  TelegramState.UNDEFINED                : TELEGRAM_STATE_TO_STRING := StrReplace('UNDEFINED ({0})'               ,'{0}', USINT_TO_STRING(State));
  TelegramState.ERROR_161                : TELEGRAM_STATE_TO_STRING := StrReplace('ERROR_161 ({0})'               ,'{0}', USINT_TO_STRING(State));
  TelegramState.ERROR_162                : TELEGRAM_STATE_TO_STRING := StrReplace('ERROR_162 ({0})'               ,'{0}', USINT_TO_STRING(State));
  TelegramState.ERROR_163                : TELEGRAM_STATE_TO_STRING := StrReplace('ERROR_163 ({0})'               ,'{0}', USINT_TO_STRING(State));
  TelegramState.ERROR_164                : TELEGRAM_STATE_TO_STRING := StrReplace('ERROR_164 ({0})'               ,'{0}', USINT_TO_STRING(State));
  TelegramState.ERROR_165                : TELEGRAM_STATE_TO_STRING := StrReplace('ERROR_165 ({0})'               ,'{0}', USINT_TO_STRING(State));
  TelegramState.ERROR_166                : TELEGRAM_STATE_TO_STRING := StrReplace('ERROR_166 ({0})'               ,'{0}', USINT_TO_STRING(State));
  TelegramState.ERROR_167                : TELEGRAM_STATE_TO_STRING := StrReplace('ERROR_167 ({0})'               ,'{0}', USINT_TO_STRING(State));
  TelegramState.ERROR_168                : TELEGRAM_STATE_TO_STRING := StrReplace('ERROR_168 ({0})'               ,'{0}', USINT_TO_STRING(State));
  TelegramState.ERROR_169                : TELEGRAM_STATE_TO_STRING := StrReplace('ERROR_169 ({0})'               ,'{0}', USINT_TO_STRING(State));
  TelegramState.ERROR_170                : TELEGRAM_STATE_TO_STRING := StrReplace('ERROR_170 ({0})'               ,'{0}', USINT_TO_STRING(State));
  TelegramState.ERROR_171                : TELEGRAM_STATE_TO_STRING := StrReplace('ERROR_171 ({0})'               ,'{0}', USINT_TO_STRING(State));
  TelegramState.ERROR_172                : TELEGRAM_STATE_TO_STRING := StrReplace('ERROR_172 ({0})'               ,'{0}', USINT_TO_STRING(State));
  TelegramState.READY_TO_RESUME          : TELEGRAM_STATE_TO_STRING := StrReplace('READY_TO_RESUME ({0})'         ,'{0}', USINT_TO_STRING(State));
  TelegramState.READY_FOR_INITIALIZATION : TELEGRAM_STATE_TO_STRING := StrReplace('READY_FOR_INITIALIZATION ({0})','{0}', USINT_TO_STRING(State));
  TelegramState.INITIALIZED              : TELEGRAM_STATE_TO_STRING := StrReplace('INITIALIZED ({0})'             ,'{0}', USINT_TO_STRING(State));  
ELSE
  TELEGRAM_STATE_TO_STRING := CONCAT('TelegramStateToString-Function: Error -> no parsing for value ', USINT_TO_STRING(State));
END_CASE

END_FUNCTION

// Library/Functions/Convert/TO_STRING/THRESHOLD_MODE_TO_STRING
FUNCTION THRESHOLD_MODE_TO_STRING : STRING
// ------------------------------------------------------------------------- 
//  SRCI Robot Library                                                
// ------------------------------------------------------------------------- 
//                                                                           
//  Object:      THRESHOLD_MODE_TO_STRING                                       
//  Author:      Thorsten Brach                                                
//  Date:        2025-01-24
//
//  Description:                                              
//   
//                                                                           
//  Copyright: 
//    (C) 2025 Thorsten Brach. All rights reserved                                                                                                                                            
//             Licensed under the LGPL-3.0 license.
//                                                                           
//  Disclaimer:                                                                           
//    This project is provided without any guarantee and can be used for   
//    private and commercial purposes. Any use is at the user’s 
//    own risk and responsibility.
//
// -------------------------------------------------------------------------
VAR_INPUT
  /// ThresholdMode
  Value : ThresholdMode;
END_VAR

CASE Value 
OF

  ThresholdMode.AUTOMATIC : StrReplace('AUTOMATIC ({0})','{0}' , USINT_TO_STRING(Value));
  ThresholdMode.MANUAL    : StrReplace('MANUAL ({0})'   ,'{0}' , USINT_TO_STRING(Value));

END_CASE

END_FUNCTION

// Library/Functions/Convert/TO_STRING/TOOL_CALCULATION_MODE_TO_STRING
FUNCTION TOOL_CALCULATION_MODE_TO_STRING : STRING
// ------------------------------------------------------------------------- 
//  SRCI Robot Library                                                
// ------------------------------------------------------------------------- 
//                                                                           
//  Object:      TOOL_CALCULATION_MODE_TO_STRING                                       
//  Author:      Thorsten Brach                                                
//  Date:        2025-02-01
//
//  Description:                                              
//   
//                                                                           
//  Copyright: 
//    (C) 2025 Thorsten Brach. All rights reserved                                                                                                                                            
//             Licensed under the LGPL-3.0 license.
//                                                                           
//  Disclaimer:                                                                           
//    This project is provided without any guarantee and can be used for   
//    private and commercial purposes. Any use is at the user’s 
//    own risk and responsibility.
//
// -------------------------------------------------------------------------
VAR_INPUT
  /// ToolCalculationMode
  Value : ToolCalculationMode;
END_VAR

CASE Value 
OF

  ToolCalculationMode.TWO_POINT_Z_METHOD   : StrReplace('TWO_POINT_Z_METHOD ({0})'  ,'{0}' , SINT_TO_STRING(Value));
  ToolCalculationMode.THREE_POINT_METHOD   : StrReplace('THREE_POINT_METHOD ({0})'  ,'{0}' , SINT_TO_STRING(Value));
  ToolCalculationMode.FOUR_POINT_METHOD    : StrReplace('FOUR_POINT_METHOD ({0})'   ,'{0}' , SINT_TO_STRING(Value));
  ToolCalculationMode.FIVE_POINT_METHOD    : StrReplace('FIVE_POINT_METHOD ({0})'   ,'{0}' , SINT_TO_STRING(Value));
  ToolCalculationMode.SIX_POINT_METHOD     : StrReplace('SIX_POINT_METHOD ({0})'    ,'{0}' , SINT_TO_STRING(Value));
  ToolCalculationMode.ABC_WORLD_METHOD     : StrReplace('ABC_WORLD_METHOD ({0})'    ,'{0}' , SINT_TO_STRING(Value));
  ToolCalculationMode.ABC_TWO_POINT_METHOD : StrReplace('ABC_TWO_POINT_METHOD ({0})','{0}' , SINT_TO_STRING(Value));
  
END_CASE

END_FUNCTION

// Library/Functions/Convert/TO_STRING/TRANSFORM_MODE_TO_STRING
FUNCTION TRANSFORM_MODE_TO_STRING : STRING
// ------------------------------------------------------------------------- 
//  SRCI Robot Library                                                
// ------------------------------------------------------------------------- 
//                                                                           
//  Object:      TRANSFORM_MODE_TO_STRING                                       
//  Author:      Thorsten Brach                                                
//  Date:        2025-01-24
//
//  Description:                                              
//   
//                                                                           
//  Copyright: 
//    (C) 2025 Thorsten Brach. All rights reserved                                                                                                                                            
//             Licensed under the LGPL-3.0 license.
//                                                                           
//  Disclaimer:                                                                           
//    This project is provided without any guarantee and can be used for   
//    private and commercial purposes. Any use is at the user’s 
//    own risk and responsibility.
//
// -------------------------------------------------------------------------
VAR_INPUT
  /// TransformMode
  Value : TransformMode;
END_VAR

CASE Value 
OF

  TransformMode.MIRROR_AT_POINT             : StrReplace('MIRROR_AT_POINT ({0})'             ,'{0}' , SINT_TO_STRING(Value));
  TransformMode.MIRROR_AT_STRAIGHT_LINE     : StrReplace('MIRROR_AT_STRAIGHT_LINE ({0})'     ,'{0}' , SINT_TO_STRING(Value));
  TransformMode.MIRROR_AT_PLANE             : StrReplace('MIRROR_AT_PLANE ({0})'             ,'{0}' , SINT_TO_STRING(Value));
  TransformMode.ROTATE_AROUND_STRAIGHT_LINE : StrReplace('ROTATE_AROUND_STRAIGHT_LINE ({0})' ,'{0}' , SINT_TO_STRING(Value));
  TransformMode.SHIFT_BY_VECTOR             : StrReplace('SHIFT_BY_VECTOR ({0})'             ,'{0}' , SINT_TO_STRING(Value));

END_CASE

END_FUNCTION

// Library/Functions/Convert/TO_STRING/TRIGGER_CONDITION_TO_STRING
FUNCTION TRIGGER_CONDITION_TO_STRING : STRING
// ------------------------------------------------------------------------- 
//  SRCI Robot Library                                                
// ------------------------------------------------------------------------- 
//                                                                           
//  Object:      TRIGGER_CONDITION_TO_STRING                                       
//  Author:      Thorsten Brach                                                
//  Date:        2025-02-01
//
//  Description:                                              
//   
//                                                                           
//  Copyright: 
//    (C) 2025 Thorsten Brach. All rights reserved                                                                                                                                            
//             Licensed under the LGPL-3.0 license.
//                                                                           
//  Disclaimer:                                                                           
//    This project is provided without any guarantee and can be used for   
//    private and commercial purposes. Any use is at the user’s 
//    own risk and responsibility.
//
// -------------------------------------------------------------------------
VAR_INPUT
  /// TriggerCondition
  Value : TriggerCondition;
END_VAR

CASE Value 
OF

  TriggerCondition.TARGET_POSITION_TIME_MS                : StrReplace('TARGET_POSITION_TIME_MS ({0})'               ,'{0}' , SINT_TO_STRING(Value));
  TriggerCondition.TARGET_POSITION_TCP_VELOCITY_ABSOLUTE  : StrReplace('TARGET_POSITION_TCP_VELOCITY_ABSOLUTE ({0})' ,'{0}' , SINT_TO_STRING(Value));
  TriggerCondition.TARGET_POSITION_TCP_VELOCITY_PERCENT   : StrReplace('TARGET_POSITION_TCP_VELOCITY_PERCENT ({0})'  ,'{0}' , SINT_TO_STRING(Value));
  TriggerCondition.TARGET_POSITION_DISTANCE_ABSOLUTE      : StrReplace('TARGET_POSITION_DISTANCE_ABSOLUTE ({0})'     ,'{0}' , SINT_TO_STRING(Value));
  TriggerCondition.TARGET_POSITION_DISTANCE_PERCENT       : StrReplace('TARGET_POSITION_DISTANCE_PERCENT ({0})'      ,'{0}' , SINT_TO_STRING(Value));
  TriggerCondition.UNDEFINED                              : StrReplace('UNDEFINED ({0})'                             ,'{0}' , SINT_TO_STRING(Value));
  TriggerCondition.START_POSITION_DISTANCE_PERCENT        : StrReplace('START_POSITION_DISTANCE_PERCENT ({0})'       ,'{0}' , SINT_TO_STRING(Value));
  TriggerCondition.START_POSITION_DISTANCE_ABSOLUTE       : StrReplace('START_POSITION_DISTANCE_ABSOLUTE ({0})'      ,'{0}' , SINT_TO_STRING(Value));
  TriggerCondition.START_POSITION_TCP_VELOCITY_PERCENT    : StrReplace('START_POSITION_TCP_VELOCITY_PERCENT ({0})'   ,'{0}' , SINT_TO_STRING(Value));
  TriggerCondition.START_POSITION_TCP_VELOCIT_ABSOLUTE    : StrReplace('START_POSITION_TCP_VELOCIT_ABSOLUTE ({0})'   ,'{0}' , SINT_TO_STRING(Value));
  TriggerCondition.START_POSITION_TIME_MS                 : StrReplace('START_POSITION_TCP_VELOCIT_ABSOLUTE ({0})'   ,'{0}' , SINT_TO_STRING(Value));

END_CASE

END_FUNCTION

// Library/Functions/Convert/TO_STRING/TRIGGER_MODE_IO_TO_STRING
FUNCTION TRIGGER_MODE_IO_TO_STRING : STRING
// ------------------------------------------------------------------------- 
//  SRCI Robot Library                                                
// ------------------------------------------------------------------------- 
//                                                                           
//  Object:      TRIGGER_MODE_IO_TO_STRING                                       
//  Author:      Thorsten Brach                                                
//  Date:        2025-02-01
//
//  Description:                                              
//   
//                                                                           
//  Copyright: 
//    (C) 2025 Thorsten Brach. All rights reserved                                                                                                                                            
//             Licensed under the LGPL-3.0 license.
//                                                                           
//  Disclaimer:                                                                           
//    This project is provided without any guarantee and can be used for   
//    private and commercial purposes. Any use is at the user’s 
//    own risk and responsibility.
//
// -------------------------------------------------------------------------
VAR_INPUT
  /// TriggerModeIo
  Value : TriggerModeIo;
END_VAR

CASE Value 
OF

  TriggerModeIo.INVALID                                                             : StrReplace('INVALID ({0})'                                                              ,'{0}' , SINT_TO_STRING(Value));
  TriggerModeIo.DIGITAL_INPUT_RISING_EDGE                                           : StrReplace('DIGITAL_INPUT_RISING_EDGE ({0})'                                            ,'{0}' , SINT_TO_STRING(Value));
  TriggerModeIo.DIGITAL_INPUT_FALLING_EDGE                                          : StrReplace('DIGITAL_INPUT_FALLING_EDGE ({0})'                                           ,'{0}' , SINT_TO_STRING(Value));
  TriggerModeIo.DIGITAL_INPUT_RISING_OR_FALLING_EDGE                                : StrReplace('DIGITAL_INPUT_RISING_OR_FALLING_EDGE ({0})'                                 ,'{0}' , SINT_TO_STRING(Value));
  TriggerModeIo.DIGITAL_INPUT_RISING_OR_FALLING_EDGE_INVERTED                       : StrReplace('DIGITAL_INPUT_RISING_OR_FALLING_EDGE_INVERTED ({0})'                        ,'{0}' , SINT_TO_STRING(Value));
  TriggerModeIo.DIGITAL_OUTPUT_RISING_EDGE                                          : StrReplace('DIGITAL_OUTPUT_RISING_EDGE ({0})'                                           ,'{0}' , SINT_TO_STRING(Value));
  TriggerModeIo.DIGITAL_OUTPUT_FALLING_EDGE                                         : StrReplace('DIGITAL_OUTPUT_FALLING_EDGE ({0})'                                          ,'{0}' , SINT_TO_STRING(Value));
  TriggerModeIo.DIGITAL_OUTPUT_RISING_OR_FALLING_EDGE                               : StrReplace('DIGITAL_OUTPUT_RISING_OR_FALLING_EDGE ({0})'                                ,'{0}' , SINT_TO_STRING(Value));
  TriggerModeIo.DIGITAL_OUTPUT_RISING_OR_FALLING_EDGE_INVERTED                      : StrReplace('DIGITAL_OUTPUT_RISING_OR_FALLING_EDGE_INVERTED ({0})'                       ,'{0}' , SINT_TO_STRING(Value));
  TriggerModeIo.ANALOG_INPUT_EXCEEDING_DEFINED_THRESHOLD                            : StrReplace('ANALOG_INPUT_EXCEEDING_DEFINED_THRESHOLD ({0})'                             ,'{0}' , SINT_TO_STRING(Value));
  TriggerModeIo.ANALOG_INPUT_FALLING_BELOW_DEFINED_THRESHOLD                        : StrReplace('ANALOG_INPUT_FALLING_BELOW_DEFINED_THRESHOLD ({0})'                         ,'{0}' , SINT_TO_STRING(Value));
  TriggerModeIo.ANALOG_INPUT_EXCEEDING_OR_FALLING_BELOW_DEFINED_THRESHOLD           : StrReplace('ANALOG_INPUT_EXCEEDING_OR_FALLING_BELOW_DEFINED_THRESHOLD ({0})'            ,'{0}' , SINT_TO_STRING(Value));
  TriggerModeIo.ANALOG_INPUT_EXCEEDING_OR_FALLING_BELOW_DEFINED_THRESHOLD_INVERTED  : StrReplace('ANALOG_INPUT_EXCEEDING_OR_FALLING_BELOW_DEFINED_THRESHOLD_INVERTED ({0})'   ,'{0}' , SINT_TO_STRING(Value));
  TriggerModeIo.ANALOG_INPUT_ENTERING_DEFINED_RANGE                                 : StrReplace('ANALOG_INPUT_ENTERING_DEFINED_RANGE ({0})'                                  ,'{0}' , SINT_TO_STRING(Value));
  TriggerModeIo.ANALOG_INPUT_LEAVING_DEFINED_RANGE                                  : StrReplace('ANALOG_INPUT_LEAVING_DEFINED_RANGE ({0})'                                   ,'{0}' , SINT_TO_STRING(Value));
  TriggerModeIo.ANALOG_INPUT_ENTERING_OR_LEAVING_DEFINED_RANGE                      : StrReplace('ANALOG_INPUT_ENTERING_OR_LEAVING_DEFINED_RANGE ({0})'                       ,'{0}' , SINT_TO_STRING(Value));
  TriggerModeIo.ANALOG_INPUT_ENTERING_OR_LEAVING_DEFINED_RANGE_INVERTED             : StrReplace('ANALOG_INPUT_ENTERING_OR_LEAVING_DEFINED_RANGE_INVERTED ({0})'              ,'{0}' , SINT_TO_STRING(Value));
  TriggerModeIo.ANALOG_OUTPUT_EXCEEDING_DEFINED_THRESHOLD                           : StrReplace('ANALOG_OUTPUT_EXCEEDING_DEFINED_THRESHOLD ({0})'                            ,'{0}' , SINT_TO_STRING(Value));
  TriggerModeIo.ANALOG_OUTPUT_FALLING_BELOW_DEFINED_THRESHOLD                       : StrReplace('ANALOG_OUTPUT_FALLING_BELOW_DEFINED_THRESHOLD ({0})'                        ,'{0}' , SINT_TO_STRING(Value));
  TriggerModeIo.ANALOG_OUTPUT_EXCEEDING_OR_FALLING_BELOW_DEFINED_THRESHOLD          : StrReplace('ANALOG_OUTPUT_EXCEEDING_OR_FALLING_BELOW_DEFINED_THRESHOLD ({0})'           ,'{0}' , SINT_TO_STRING(Value));
  TriggerModeIo.ANALOG_OUTPUT_EXCEEDING_OR_FALLING_BELOW_DEFINED_THRESHOLD_INVERTED : StrReplace('ANALOG_OUTPUT_EXCEEDING_OR_FALLING_BELOW_DEFINED_THRESHOLD_INVERTED ({0})'  ,'{0}' , SINT_TO_STRING(Value));
  TriggerModeIo.ANALOG_OUTPUT_ENTERING_DEFINED_RANGE                                : StrReplace('ANALOG_OUTPUT_ENTERING_DEFINED_RANGE ({0})'                                 ,'{0}' , SINT_TO_STRING(Value));
  TriggerModeIo.ANALOG_OUTPUT_LEAVING_DEFINED_RANGE                                 : StrReplace('ANALOG_OUTPUT_LEAVING_DEFINED_RANGE ({0})'                                  ,'{0}' , SINT_TO_STRING(Value));
  TriggerModeIo.ANALOG_OUTPUT_ENTERING_OR_LEAVING_DEFINED_RANGE                     : StrReplace('ANALOG_OUTPUT_ENTERING_OR_LEAVING_DEFINED_RANGE ({0})'                      ,'{0}' , SINT_TO_STRING(Value));
  TriggerModeIo.ANALOG_OUTPUT_ENTERING_OR_LEAVING_DEFINED_RANGE_INVERTED            : StrReplace('ANALOG_OUTPUT_ENTERING_OR_LEAVING_DEFINED_RANGE_INVERTED ({0})'             ,'{0}' , SINT_TO_STRING(Value));
  TriggerModeIo.INTEGER_REGISTER_EXCEEDING_DEFINED_THRESHOLD                        : StrReplace('INTEGER_REGISTER_EXCEEDING_DEFINED_THRESHOLD ({0})'                         ,'{0}' , SINT_TO_STRING(Value));
  TriggerModeIo.INTEGER_REGISTER_FALLING_BELOW_DEFINED_THRESHOLD                    : StrReplace('INTEGER_REGISTER_FALLING_BELOW_DEFINED_THRESHOLD ({0})'                     ,'{0}' , SINT_TO_STRING(Value));
  TriggerModeIo.INTEGER_REGISTER_EXCEEDING_OR_FALLING_BELOW_DEFINED_THRESHOLD       : StrReplace('INTEGER_REGISTER_EXCEEDING_OR_FALLING_BELOW_DEFINED_THRESHOLD ({0})'        ,'{0}' , SINT_TO_STRING(Value));
  TriggerModeIo.INTEGER_REGISTER_EXCEEDING_OR_FALLING_BELOW_DEFINED_VALUE_INVERTED  : StrReplace('INTEGER_REGISTER_EXCEEDING_OR_FALLING_BELOW_DEFINED_VALUE_INVERTED ({0})'   ,'{0}' , SINT_TO_STRING(Value));
  TriggerModeIo.INTEGER_REGISTER_ENTERING_DEFINED_RANGE                             : StrReplace('INTEGER_REGISTER_ENTERING_DEFINED_RANGE ({0})'                              ,'{0}' , SINT_TO_STRING(Value));
  TriggerModeIo.INTEGER_REGISTER_LEAVING_DEFINED_RANGE                              : StrReplace('INTEGER_REGISTER_LEAVING_DEFINED_RANGE ({0})'                               ,'{0}' , SINT_TO_STRING(Value));
  TriggerModeIo.INTEGER_REGISTER_ENTERING_OR_LEAVING_DEFINED_RANGE                  : StrReplace('INTEGER_REGISTER_ENTERING_OR_LEAVING_DEFINED_RANGE ({0})'                   ,'{0}' , SINT_TO_STRING(Value));
  TriggerModeIo.INTEGER_REGISTER_ENTERING_OR_LEAVING_DEFINED_RANGE_INVERTED         : StrReplace('INTEGER_REGISTER_ENTERING_OR_LEAVING_DEFINED_RANGE_INVERTED ({0})'          ,'{0}' , SINT_TO_STRING(Value));
  TriggerModeIo.REAL_REGISTER_EXCEEDING_DEFINED_THRESHOLD                           : StrReplace('REAL_REGISTER_EXCEEDING_DEFINED_THRESHOLD ({0})'                            ,'{0}' , SINT_TO_STRING(Value));
  TriggerModeIo.REAL_REGISTER_FALLING_BELOW_DEFINED_THRESHOLD                       : StrReplace('REAL_REGISTER_FALLING_BELOW_DEFINED_THRESHOLD ({0})'                        ,'{0}' , SINT_TO_STRING(Value));
  TriggerModeIo.REAL_REGISTER_EXCEEDING_OR_FALLING_BELOW_DEFINED_THRESHOLD          : StrReplace('REAL_REGISTER_EXCEEDING_OR_FALLING_BELOW_DEFINED_THRESHOLD ({0})'           ,'{0}' , SINT_TO_STRING(Value));
  TriggerModeIo.REAL_REGISTER_EXCEEDING_OR_FALLING_BELOW_DEFINED_THRESHOLD_INVERTED : StrReplace('REAL_REGISTER_EXCEEDING_OR_FALLING_BELOW_DEFINED_THRESHOLD_INVERTED ({0})'  ,'{0}' , SINT_TO_STRING(Value));
  TriggerModeIo.REAL_REGISTER_ENTERING_DEFINED_RANGE                                : StrReplace('REAL_REGISTER_ENTERING_DEFINED_RANGE ({0})'                                 ,'{0}' , SINT_TO_STRING(Value));
  TriggerModeIo.REAL_REGISTER_LEAVING_DEFINED_RANGE                                 : StrReplace('REAL_REGISTER_LEAVING_DEFINED_RANGE ({0})'                                  ,'{0}' , SINT_TO_STRING(Value));
  TriggerModeIo.REAL_REGISTER_ENTERING_OR_LEAVING_DEFINED_RANGE                     : StrReplace('REAL_REGISTER_ENTERING_OR_LEAVING_DEFINED_RANGE ({0})'                      ,'{0}' , SINT_TO_STRING(Value));
  TriggerModeIo.REAL_REGISTER_ENTERING_OR_LEAVING_DEFINED_RANGE_INVERTED            : StrReplace('REAL_REGISTER_ENTERING_OR_LEAVING_DEFINED_RANGE_INVERTED ({0})'             ,'{0}' , SINT_TO_STRING(Value));
END_CASE

END_FUNCTION

// Library/Functions/Convert/TO_STRING/TRIGGER_MODE_MEASUREMENT_TO_STRING
FUNCTION TRIGGER_MODE_MEASUREMENT_TO_STRING : STRING
// ------------------------------------------------------------------------- 
//  SRCI Robot Library                                                
// ------------------------------------------------------------------------- 
//                                                                           
//  Object:      TRIGGER_MODE_MEASUREMENT_TO_STRING                                       
//  Author:      Thorsten Brach                                                
//  Date:        2025-01-24
//
//  Description:                                              
//   
//                                                                           
//  Copyright: 
//    (C) 2025 Thorsten Brach. All rights reserved                                                                                                                                            
//             Licensed under the LGPL-3.0 license.
//                                                                           
//  Disclaimer:                                                                           
//    This project is provided without any guarantee and can be used for   
//    private and commercial purposes. Any use is at the user’s 
//    own risk and responsibility.
//
// -------------------------------------------------------------------------
VAR_INPUT
  /// TriggerMode
  Value : TriggerModeMeasurement;
END_VAR

CASE Value 
OF

  TriggerModeMeasurement.NO_TRIGGER                   : StrReplace('NO_TRIGGER ({0})'                   ,'{0}' , USINT_TO_STRING(Value));
  TriggerModeMeasurement.POSITIVE_START_NEGATIVE_STOP : StrReplace('POSITIVE_START_NEGATIVE_STOP ({0})' ,'{0}' , USINT_TO_STRING(Value));
  TriggerModeMeasurement.POSITIVE_START_STOP          : StrReplace('POSITIVE_START_STOP ({0})'          ,'{0}' , USINT_TO_STRING(Value));

END_CASE

END_FUNCTION

// Library/Functions/Convert/TO_STRING/TRIGGER_REACTION_MODE_TO_STRING
FUNCTION TRIGGER_REACTION_MODE_TO_STRING : STRING
// ------------------------------------------------------------------------- 
//  SRCI Robot Library                                                
// ------------------------------------------------------------------------- 
//                                                                           
//  Object:      TRIGGER_REACTION_MODE_TO_STRING                                       
//  Author:      Thorsten Brach                                                
//  Date:        2025-02-01
//
//  Description:                                              
//   
//                                                                           
//  Copyright: 
//    (C) 2025 Thorsten Brach. All rights reserved                                                                                                                                            
//             Licensed under the LGPL-3.0 license.
//                                                                           
//  Disclaimer:                                                                           
//    This project is provided without any guarantee and can be used for   
//    private and commercial purposes. Any use is at the user’s 
//    own risk and responsibility.
//
// -------------------------------------------------------------------------
VAR_INPUT
  /// TriggerReactionMode
  Value : TriggerReactionMode;
END_VAR

CASE Value 
OF

  TriggerReactionMode.NO_REACTION                : StrReplace('NO_REACTION ({0})'                 ,'{0}' , SINT_TO_STRING(Value));
  TriggerReactionMode.INTERRUPT                  : StrReplace('INTERRUPT ({0})'                   ,'{0}' , SINT_TO_STRING(Value));
  TriggerReactionMode.GROUP_STOP                 : StrReplace('GROUP_STOP ({0})'                  ,'{0}' , SINT_TO_STRING(Value));
  TriggerReactionMode.DISABLE_ROBOT              : StrReplace('DISABLE_ROBOT ({0})'               ,'{0}' , SINT_TO_STRING(Value));
  TriggerReactionMode.STOP_ACTUAL_MOTION_COMMAND : StrReplace('STOP_ACTUAL_MOTION_COMMAND ({0})'  ,'{0}' , SINT_TO_STRING(Value));

END_CASE

END_FUNCTION

// Library/Functions/Convert/TO_STRING/TURN_MODE_TO_STRING
FUNCTION TURN_MODE_TO_STRING : STRING
// ------------------------------------------------------------------------- 
//  SRCI Robot Library                                                
// ------------------------------------------------------------------------- 
//                                                                           
//  Object:      TURN_MODE_TO_STRING                                       
//  Author:      Thorsten Brach                                                
//  Date:        2025-01-23
//
//  Description:                                              
//   
//                                                                           
//  Copyright: 
//    (C) 2025 Thorsten Brach. All rights reserved                                                                                                                                            
//             Licensed under the LGPL-3.0 license.
//                                                                           
//  Disclaimer:                                                                           
//    This project is provided without any guarantee and can be used for   
//    private and commercial purposes. Any use is at the user’s 
//    own risk and responsibility.
//
// -------------------------------------------------------------------------
VAR_INPUT
  /// TurnMode
  Value : TurnMode;
END_VAR

CASE Value 
OF

  TurnMode.USE_TURN_NUMBER : StrReplace('USE_TURN_NUMBER ({0})','{0}' , USINT_TO_STRING(Value));
  TurnMode.SAME            : StrReplace('SAME ({0})'           ,'{0}' , USINT_TO_STRING(Value));
  TurnMode.FREE            : StrReplace('FREE ({0})'           ,'{0}' , USINT_TO_STRING(Value));

END_CASE

END_FUNCTION

// Library/Functions/Convert/TO_STRING/WORD_TO_STRING_BIN
FUNCTION WORD_TO_STRING_BIN : STRING
// ------------------------------------------------------------------------- 
//  SRCI Robot Library                                                
// ------------------------------------------------------------------------- 
//                                                                           
//  Object:      WORD_TO_STRING_BIN                                       
//  Author:      Thorsten Brach                                                
//  Date:        2025-02-03
//
//  Description:                                              
//    Converts a BYTE to a STRING with binary notation  
//                                                                           
//  Copyright: 
//    (C) 2024 Thorsten Brach. All rights reserved                                                                                                                                            
//             Licensed under the LGPL-3.0 license.
//                                                                           
//  Disclaimer:                                                                           
//    This project is provided without any guarantee and can be used for   
//    private and commercial purposes. Any use is at the user’s 
//    own risk and responsibility.
//
// -------------------------------------------------------------------------
VAR_INPUT
 /// Value to convert
 Value : WORD; 
END_VAR

WORD_TO_STRING_BIN := '2#';

IF (Value.15)
THEN
  WORD_TO_STRING_BIN := CONCAT(WORD_TO_STRING_BIN, '1');
ELSE
  WORD_TO_STRING_BIN := CONCAT(WORD_TO_STRING_BIN, '0');
END_IF

IF (Value.14)
THEN
  WORD_TO_STRING_BIN := CONCAT(WORD_TO_STRING_BIN, '1');
ELSE
  WORD_TO_STRING_BIN := CONCAT(WORD_TO_STRING_BIN, '0');
END_IF

IF (Value.13)
THEN
  WORD_TO_STRING_BIN := CONCAT(WORD_TO_STRING_BIN, '1');
ELSE
  WORD_TO_STRING_BIN := CONCAT(WORD_TO_STRING_BIN, '0');
END_IF

IF (Value.12)
THEN
  WORD_TO_STRING_BIN := CONCAT(WORD_TO_STRING_BIN, '1_');
ELSE
  WORD_TO_STRING_BIN := CONCAT(WORD_TO_STRING_BIN, '0_');
END_IF

IF (Value.11)
THEN
  WORD_TO_STRING_BIN := CONCAT(WORD_TO_STRING_BIN, '1');
ELSE
  WORD_TO_STRING_BIN := CONCAT(WORD_TO_STRING_BIN, '0');
END_IF

IF (Value.10)
THEN
  WORD_TO_STRING_BIN := CONCAT(WORD_TO_STRING_BIN, '1');
ELSE
  WORD_TO_STRING_BIN := CONCAT(WORD_TO_STRING_BIN, '0');
END_IF

IF (Value.09)
THEN
  WORD_TO_STRING_BIN := CONCAT(WORD_TO_STRING_BIN, '1');
ELSE
  WORD_TO_STRING_BIN := CONCAT(WORD_TO_STRING_BIN, '0');
END_IF

IF (Value.08)
THEN
  WORD_TO_STRING_BIN := CONCAT(WORD_TO_STRING_BIN, '1_');
ELSE
  WORD_TO_STRING_BIN := CONCAT(WORD_TO_STRING_BIN, '0_');
END_IF

IF (Value.7)
THEN
  WORD_TO_STRING_BIN := CONCAT(WORD_TO_STRING_BIN, '1');
ELSE
  WORD_TO_STRING_BIN := CONCAT(WORD_TO_STRING_BIN, '0');
END_IF

IF (Value.6)
THEN
  WORD_TO_STRING_BIN := CONCAT(WORD_TO_STRING_BIN, '1');
ELSE
  WORD_TO_STRING_BIN := CONCAT(WORD_TO_STRING_BIN, '0');
END_IF

IF (Value.5)
THEN
  WORD_TO_STRING_BIN := CONCAT(WORD_TO_STRING_BIN, '1');
ELSE
  WORD_TO_STRING_BIN := CONCAT(WORD_TO_STRING_BIN, '0');
END_IF

IF (Value.4)
THEN
  WORD_TO_STRING_BIN := CONCAT(WORD_TO_STRING_BIN, '1_');
ELSE
  WORD_TO_STRING_BIN := CONCAT(WORD_TO_STRING_BIN, '0_');
END_IF

IF (Value.3)
THEN
  WORD_TO_STRING_BIN := CONCAT(WORD_TO_STRING_BIN, '1');
ELSE
  WORD_TO_STRING_BIN := CONCAT(WORD_TO_STRING_BIN, '0');
END_IF

IF (Value.2)
THEN
  WORD_TO_STRING_BIN := CONCAT(WORD_TO_STRING_BIN, '1');
ELSE
  WORD_TO_STRING_BIN := CONCAT(WORD_TO_STRING_BIN, '0');
END_IF

IF (Value.1)
THEN
  WORD_TO_STRING_BIN := CONCAT(WORD_TO_STRING_BIN, '1');
ELSE
  WORD_TO_STRING_BIN := CONCAT(WORD_TO_STRING_BIN, '0');
END_IF


IF (Value.0)
THEN
  WORD_TO_STRING_BIN := CONCAT(WORD_TO_STRING_BIN, '1');
ELSE
  WORD_TO_STRING_BIN := CONCAT(WORD_TO_STRING_BIN, '0');
END_IF


WORD_TO_STRING_BIN := CONCAT(WORD_TO_STRING_BIN, ' (');
WORD_TO_STRING_BIN := CONCAT(WORD_TO_STRING_BIN, WORD_TO_STRING(Value));
WORD_TO_STRING_BIN := CONCAT(WORD_TO_STRING_BIN, ')');

END_FUNCTION

// Library/Functions/Convert/TO_STRING/WORD_TO_STRING_HEX
FUNCTION WORD_TO_STRING_HEX : STRING
// ------------------------------------------------------------------------- 
//  SRCI Robot Library                                                
// ------------------------------------------------------------------------- 
//                                                                           
//  Object:      WORD_TO_STRING_HEX                                       
//  Author:      Thorsten Brach                                                
//  Date:        2024-12-13
//
//  Description:                                              
//    Converts a WORD to a STRING with hex notation  
//                                                                           
//  Copyright: 
//    (C) 2024 Thorsten Brach. All rights reserved                                                                                                                                            
//             Licensed under the LGPL-3.0 license.
//                                                                           
//  Disclaimer:                                                                           
//    This project is provided without any guarantee and can be used for   
//    private and commercial purposes. Any use is at the user’s 
//    own risk and responsibility.
//
// -------------------------------------------------------------------------
VAR_INPUT
 /// Value to convert
 Value : WORD; 
END_VAR
VAR
  /// high Byte
 _highByte   : BYTE;      
  /// low Byte
 _lowByte    : BYTE;      
  /// high Nibble
 _highNibble : BYTE;     
  /// low Nibble 
 _lowNibble  : BYTE;     
  /// single Hex char
  hexChar    : STRING(1);
  /// Hex chars  
  hexChars   : ARRAY[0..15] OF STRING(1) := ['0', '1', '2', '3', '4', '5', '6', '7', '8', '9', 'A', 'B', 'C', 'D', 'E', 'F'];
END_VAR

// get high and low byte from word
_highByte := WORD_TO_BYTE(SHR(Value, 8)); 
_lowByte  := WORD_TO_BYTE(Value AND 16#FF); 

// convert highest Byte to HEX
_highNibble := SHR(_highByte, 4);   
_lowNibble  := (_highByte AND 16#F);
WORD_TO_STRING_HEX := CONCAT(hexChars[_highNibble], hexChars[_lowNibble]);

// convert lowest Byte to HEX
_highNibble := SHR(_lowByte, 4); 
_lowNibble := _lowByte AND 16#F; 
WORD_TO_STRING_HEX := CONCAT(WORD_TO_STRING_HEX, CONCAT(hexChars[_highNibble], hexChars[_lowNibble]));

END_FUNCTION

// Library/Functions/Convert/TO_STRING/WORK_AREA_REACTION_MODE_TO_STRING
FUNCTION WORK_AREA_REACTION_MODE_TO_STRING : STRING
// ------------------------------------------------------------------------- 
//  SRCI Robot Library                                                
// ------------------------------------------------------------------------- 
//                                                                           
//  Object:      WORK_AREA_REACTION_MODE_TO_STRING                                       
//  Author:      Thorsten Brach                                                
//  Date:        2025-02-01
//
//  Description:                                              
//   
//                                                                           
//  Copyright: 
//    (C) 2025 Thorsten Brach. All rights reserved                                                                                                                                            
//             Licensed under the LGPL-3.0 license.
//                                                                           
//  Disclaimer:                                                                           
//    This project is provided without any guarantee and can be used for   
//    private and commercial purposes. Any use is at the user’s 
//    own risk and responsibility.
//
// -------------------------------------------------------------------------
VAR_INPUT
  /// WorkAreaReactionMode
  Value : WorkAreaReactionMode;
END_VAR

CASE Value 
OF

  WorkAreaReactionMode.NO_REACTION : StrReplace('NO_REACTION ({0})','{0}' , USINT_TO_STRING(Value));
  WorkAreaReactionMode.ABORT       : StrReplace('ABORT ({0})'      ,'{0}' , USINT_TO_STRING(Value));
  WorkAreaReactionMode.INTERRUPT   : StrReplace('INTERRUPT ({0})'  ,'{0}' , USINT_TO_STRING(Value));

END_CASE

END_FUNCTION

// Library/Functions/String/StrPadRight
/// Returns the given string, filled up on the right side to the given total length with the given substring
FUNCTION StrPadRight : STRING(255)
// ------------------------------------------------------------------------- 
//  SRCI Robot Library                                                
// ------------------------------------------------------------------------- 
//                                                                           
//  Object:      SwapBytes                                       
//  Author:      Thorsten Brach                                                
//  Date:        2024-12-18
//
//  Description:                                              
//   
//                                                                           
//  Copyright: 
//    (C) 2024 Thorsten Brach. All rights reserved                                                                                                                                            
//             Licensed under the LGPL-3.0 license.
//                                                                           
//  Disclaimer:                                                                           
//    This project is provided without any guarantee and can be used for   
//    private and commercial purposes. Any use is at the user’s 
//    own risk and responsibility.
//
// -------------------------------------------------------------------------
VAR_INPUT
  /// content string
  Str    : STRING(255);
  /// sub string
  SubStr : STRING(255);
  /// Length
  Length : INT; 
END_VAR

WHILE(LEN(Str) < Length)
DO
 Str := CONCAT(Str, SubStr);
END_WHILE

StrPadRight := Str;

END_FUNCTION

// Library/Functions/Swap/GetHalfeByteHi
FUNCTION GetHalfeByteHi : BYTE
// ------------------------------------------------------------------------- 
//  SRCI Robot Library                                                
// ------------------------------------------------------------------------- 
//                                                                           
//  Object:      SwapBytes                                       
//  Author:      Thorsten Brach                                                
//  Date:        2024-12-18
//
//  Description:                                              
//   
//                                                                           
//  Copyright: 
//    (C) 2024 Thorsten Brach. All rights reserved                                                                                                                                            
//             Licensed under the LGPL-3.0 license.
//                                                                           
//  Disclaimer:                                                                           
//    This project is provided without any guarantee and can be used for   
//    private and commercial purposes. Any use is at the user’s 
//    own risk and responsibility.
//
// -------------------------------------------------------------------------
VAR_INPUT
  /// Increase payload pointer 
  Value : BYTE;
END_VAR

GetHalfeByteHi.0 := Value.4;
GetHalfeByteHi.1 := Value.5;
GetHalfeByteHi.2 := Value.6;
GetHalfeByteHi.3 := Value.7;

END_FUNCTION

// Library/Functions/Swap/GetHalfeByteLo
FUNCTION GetHalfeByteLo : BYTE
// ------------------------------------------------------------------------- 
//  SRCI Robot Library                                                
// ------------------------------------------------------------------------- 
//                                                                           
//  Object:      SwapBytes                                       
//  Author:      Thorsten Brach                                                
//  Date:        2024-12-18
//
//  Description:                                              
//   
//                                                                           
//  Copyright: 
//    (C) 2024 Thorsten Brach. All rights reserved                                                                                                                                            
//             Licensed under the LGPL-3.0 license.
//                                                                           
//  Disclaimer:                                                                           
//    This project is provided without any guarantee and can be used for   
//    private and commercial purposes. Any use is at the user’s 
//    own risk and responsibility.
//
// -------------------------------------------------------------------------
VAR_INPUT
  /// Increase payload pointer 
  Value : BYTE;
END_VAR

GetHalfeByteLo.0 := Value.0;
GetHalfeByteLo.1 := Value.1;
GetHalfeByteLo.2 := Value.2;
GetHalfeByteLo.3 := Value.3;

END_FUNCTION

// Library/Functions/Swap/SwapDword
FUNCTION SwapDword : DWORD
// ------------------------------------------------------------------------- 
//  SRCI Robot Library                                                
// ------------------------------------------------------------------------- 
//                                                                           
//  Object:      SwapDword                                       
//  Author:      Thorsten Brach                                                
//  Date:        2024-06-01
//
//  Description:                                              
//   
//                                                                           
//  Copyright: 
//    (C) 2024 Thorsten Brach. All rights reserved                                                                                                                                            
//             Licensed under the LGPL-3.0 license.
//                                                                           
//  Disclaimer:                                                                           
//    This project is provided without any guarantee and can be used for   
//    private and commercial purposes. Any use is at the user’s 
//    own risk and responsibility.
//
// -------------------------------------------------------------------------
VAR_INPUT
  /// Value
  Value : DWORD;
END_VAR

SwapBytes(ADR(Value),SIZEOF(Value));

SwapDword := Value;

END_FUNCTION

// Library/Functions/Swap/SwapIecDate
FUNCTION SwapIecDate : IEC_DATE
// ------------------------------------------------------------------------- 
//  SRCI Robot Library                                                
// ------------------------------------------------------------------------- 
//                                                                           
//  Object:      SwapIecDate                                       
//  Author:      Thorsten Brach                                                
//  Date:        2024-06-09
//
//  Description:                                              
//   
//                                                                           
//  Copyright: 
//    (C) 2024 Thorsten Brach. All rights reserved                                                                                                                                            
//             Licensed under the LGPL-3.0 license.
//                                                                           
//  Disclaimer:                                                                           
//    This project is provided without any guarantee and can be used for   
//    private and commercial purposes. Any use is at the user’s 
//    own risk and responsibility.
//
// -------------------------------------------------------------------------
VAR_INPUT
  /// Value to swap
  Value : IEC_DATE;
END_VAR

SwapBytes(ADR(Value),SIZEOF(Value));

SwapIecDate := Value;

END_FUNCTION

// Library/Functions/Swap/SwapIecTime
FUNCTION SwapIecTime : TOD
// ------------------------------------------------------------------------- 
//  SRCI Robot Library                                                
// ------------------------------------------------------------------------- 
//                                                                           
//  Object:      SwapTime                                       
//  Author:      Thorsten Brach                                                
//  Date:        2024-06-01
//
//  Description:                                              
//   
//                                                                           
//  Copyright: 
//    (C) 2024 Thorsten Brach. All rights reserved                                                                                                                                            
//             Licensed under the LGPL-3.0 license.
//                                                                           
//  Disclaimer:                                                                           
//    This project is provided without any guarantee and can be used for   
//    private and commercial purposes. Any use is at the user’s 
//    own risk and responsibility.
//
// -------------------------------------------------------------------------
VAR_INPUT
  /// Value
  Value : TOD;
END_VAR

SwapBytes(ADR(Value),SIZEOF(Value));

SwapIecTime := Value;

END_FUNCTION

// Library/Functions/Swap/SwapInt
FUNCTION SwapInt : INT
// ------------------------------------------------------------------------- 
//  SRCI Robot Library                                                
// ------------------------------------------------------------------------- 
//                                                                           
//  Object:      SwapInt                                       
//  Author:      Thorsten Brach                                                
//  Date:        2024-06-01
//
//  Description:                                              
//   
//                                                                           
//  Copyright: 
//    (C) 2024 Thorsten Brach. All rights reserved                                                                                                                                            
//             Licensed under the LGPL-3.0 license.
//                                                                           
//  Disclaimer:                                                                           
//    This project is provided without any guarantee and can be used for   
//    private and commercial purposes. Any use is at the user’s 
//    own risk and responsibility.
//
// -------------------------------------------------------------------------
VAR_INPUT
  /// Value to swap
  Value : INT;
END_VAR

SwapBytes(ADR(Value),SIZEOF(Value));

SwapInt := Value;

END_FUNCTION

// Library/Functions/Swap/SwapReal
FUNCTION SwapReal : REAL
// ------------------------------------------------------------------------- 
//  SRCI Robot Library                                                
// ------------------------------------------------------------------------- 
//                                                                           
//  Object:      SwapReal                                       
//  Author:      Thorsten Brach                                                
//  Date:        2024-06-01
//
//  Description:                                              
//   
//                                                                           
//  Copyright: 
//    (C) 2024 Thorsten Brach. All rights reserved                                                                                                                                            
//             Licensed under the LGPL-3.0 license.
//                                                                           
//  Disclaimer:                                                                           
//    This project is provided without any guarantee and can be used for   
//    private and commercial purposes. Any use is at the user’s 
//    own risk and responsibility.
//
// -------------------------------------------------------------------------
VAR_INPUT
  /// Value
  Value : REAL;
END_VAR

SwapBytes(ADR(Value),SIZEOF(Value));

SwapReal := Value;

END_FUNCTION

// Library/Functions/Swap/SwapUdint
FUNCTION SwapUdint : UDINT
// ------------------------------------------------------------------------- 
//  SRCI Robot Library                                                
// ------------------------------------------------------------------------- 
//                                                                           
//  Object:      SwapUdint                                       
//  Author:      Thorsten Brach                                                
//  Date:        2024-06-01
//
//  Description:                                              
//   
//                                                                           
//  Copyright: 
//    (C) 2024 Thorsten Brach. All rights reserved                                                                                                                                            
//             Licensed under the LGPL-3.0 license.
//                                                                           
//  Disclaimer:                                                                           
//    This project is provided without any guarantee and can be used for   
//    private and commercial purposes. Any use is at the user’s 
//    own risk and responsibility.
//
// -------------------------------------------------------------------------
VAR_INPUT
  /// Value
  Value : UDINT;
END_VAR

SwapBytes(ADR(Value),SIZEOF(Value));

SwapUdint := Value;

END_FUNCTION

// Library/Functions/Swap/SwapUint
FUNCTION SwapUint : UINT
// ------------------------------------------------------------------------- 
//  SRCI Robot Library                                                
// ------------------------------------------------------------------------- 
//                                                                           
//  Object:      SwapUint                                       
//  Author:      Thorsten Brach                                                
//  Date:        2024-06-01
//
//  Description:                                              
//   
//                                                                           
//  Copyright: 
//    (C) 2024 Thorsten Brach. All rights reserved                                                                                                                                            
//             Licensed under the LGPL-3.0 license.
//                                                                           
//  Disclaimer:                                                                           
//    This project is provided without any guarantee and can be used for   
//    private and commercial purposes. Any use is at the user’s 
//    own risk and responsibility.
//
// -------------------------------------------------------------------------
VAR_INPUT
  /// Value to swap
  Value : UINT;
END_VAR

SwapBytes(ADR(Value),SIZEOF(Value));

SwapUint := Value;

END_FUNCTION

// Library/Functions/Swap/SwapWord
FUNCTION SwapWord : WORD
// ------------------------------------------------------------------------- 
//  SRCI Robot Library                                                
// ------------------------------------------------------------------------- 
//                                                                           
//  Object:      SwapWord                                       
//  Author:      Thorsten Brach                                                
//  Date:        2024-06-01
//
//  Description:                                              
//   
//                                                                           
//  Copyright: 
//    (C) 2024 Thorsten Brach. All rights reserved                                                                                                                                            
//             Licensed under the LGPL-3.0 license.
//                                                                           
//  Disclaimer:                                                                           
//    This project is provided without any guarantee and can be used for   
//    private and commercial purposes. Any use is at the user’s 
//    own risk and responsibility.
//
// -------------------------------------------------------------------------
VAR_INPUT
  /// Value to swap
  Value : UINT;
END_VAR

SwapBytes(ADR(Value),SIZEOF(Value));

SwapWord := Value;

END_FUNCTION

// Library/Interfaces/IMessageLogger
INTERFACE IMessageLogger

METHOD AddMessageLog
VAR_INPUT
  /// Message to add to the log
  MessageLog : AlarmMessage;
END_VAR
END_METHOD

METHOD AddSystemLog
VAR_INPUT
  /// System messafe to add to the log
  SystemLog : STRING(255);
END_VAR
END_METHOD

END_INTERFACE

// Library/Interfaces/IRobotLibraryCommandFB
INTERFACE IRobotLibraryCommandFB

METHOD PUBLIC CallBack : DINT
VAR_INPUT
  /// Response data
  RspData : AxesGroupAcyclicAcrEntryRspBuffer;  
END_VAR
END_METHOD

PROPERTY CommandData : RobotLibrarySendDataFB
GET
END_GET
SET
END_SET
END_PROPERTY

END_INTERFACE

// Library/POUs/_internal/RobotLibrarySendDataFB
{attribute 'pack_mode' := '1'} 
FUNCTION_BLOCK RobotLibrarySendDataFB
// ------------------------------------------------------------------------- 
//  SRCI Robot Library                                                
// ------------------------------------------------------------------------- 
//                                                                           
//  Object:      SendData                                      
//  Author:      Thorsten Brach                                                
//  Date:        2024-06-01
//
//  Description:                                              
//    
//                                                                           
//  Copyright: 
//    (C) 2024 Thorsten Brach. All rights reserved                                                                                                                                            
//             Licensed under the LGPL-3.0 license.
//                                                                           
//  Disclaimer:                                                                           
//    This project is provided without any guarantee and can be used for   
//    private and commercial purposes. Any use is at the user’s 
//    own risk and responsibility.
//
// -------------------------------------------------------------------------
VAR_INPUT
  /// Payload
  Payload    : ARRAY [0..RobotLibraryParameter.TELEGRAM_PAYLOAD_MAX] OF BYTE;
  /// Payload length
  PayloadLen : UDINT;
  /// Payload pointer
  PayloadPtr : UDINT;
END_VAR

/// Adds a ArmConfigParameter to the payload buffer, increase the payload pointer and returns the payload lenght
METHOD AddArmConfig : UDINT
VAR_INPUT
  /// Value to add
  Value : ArmConfigParameter;
END_VAR

VAR
  /// temporary Byte
 _tmpByte : BYTE;
END_VAR
Value := Value;

_tmpByte.0 := Value.Shoulder = ArmConfigShoulder.USE_CONFIG;
_tmpByte.1 := Value.Elbow    = ArmConfigElbow   .USE_CONFIG;
_tmpByte.2 := Value.Wrist    = ArmConfigWrist   .USE_CONFIG;

AddByte(_tmpByte);
AddByte(0);

AddArmConfig := PayloadLen;
END_METHOD

/// Adds a BOOL to the payload buffer, increase the payload pointer and returns the payload lenght
METHOD AddBool : UDINT
VAR_INPUT
  /// Value to add
  Value : BOOL;
END_VAR

VAR
  /// temporary byte
 _tmpByte : BYTE := 0;
END_VAR
_tmpByte.0 := Value;
// copy data 
SysDepMemCpy(pDest := ADR(Payload[PayloadPtr]), pSrc := ADR(_tmpByte), DataLen := SIZEOF(_tmpByte));
// inc payload pointer 
PayloadPtr := PayloadPtr + SIZEOF(_tmpByte);
// return payload len
AddBool := PayloadLen := PayloadPtr;
END_METHOD

/// Adds a BYTE to the payload buffer, increase the payload pointer and returns the payload lenght
METHOD AddByte : UDINT
VAR_INPUT
  /// Value to add
  Value : BYTE;
END_VAR
Value := Value;
// copy data 
SysDepMemCpy( pDest := ADR(Payload[PayloadPtr]), pSrc := ADR(Value), DataLen := SIZEOF(Value));
// inc payload pointer 
PayloadPtr := PayloadPtr + SIZEOF(Value);
// return payload len
AddByte := PayloadLen := PayloadPtr;
END_METHOD

/// Adds a DataBlock to the payload buffer, increase the payload pointer and returns the payload lenght
METHOD AddDataBlock : UDINT
VAR_INPUT
  /// Value to add
  pValue : POINTER TO BYTE;
  /// Size of data block
  Size   : UDINT;
END_VAR
IF (pValue = 0) OR (Size = 0 )
THEN
  RETURN;
END_IF

// copy data 
SysDepMemCpy( pDest := ADR(Payload[PayloadPtr]), pSrc := pValue, DataLen := Size);
// inc payload pointer 
PayloadPtr := PayloadPtr + Size;
// return payload len
AddDataBlock := PayloadLen := PayloadPtr;
END_METHOD

/// Adds a DataInSync to the payload buffer, increase the payload pointer and returns the payload lenght
METHOD AddDataEnableSync : UDINT
VAR_INPUT
  /// Value to add
  Value : DataEnableSync;
END_VAR

VAR
  /// temporary Byte
 _tmpByte : BYTE;
END_VAR
Value := Value;

_tmpByte.0 := Value.EnableSyncTool;
_tmpByte.1 := Value.EnableSyncFrame;
_tmpByte.2 := Value.EnableSyncLoad;
_tmpByte.3 := Value.EnableSyncWorkArea;
_tmpByte.4 := Value.EnableSyncSWLimits;
_tmpByte.5 := Value.EnableSyncDefaultDynamics;
_tmpByte.6 := Value.EnableSyncReferenceDynamics;
_tmpByte.7 := Value.AllowDynamicBlending;



AddByte(_tmpByte);

AddDataEnableSync := PayloadLen;
END_METHOD

/// Adds a DataInSync to the payload buffer, increase the payload pointer and returns the payload lenght
METHOD AddDataInSync : UDINT
VAR_INPUT
  /// Value to add
  Value : DataInSync;
END_VAR

VAR
  /// temporary Byte
 _tmpByte : BYTE;
END_VAR
Value := Value;

_tmpByte.0 := Value.ToolsInSync;
_tmpByte.1 := Value.FramesInSync;
_tmpByte.2 := Value.LoadsInSync;
_tmpByte.3 := Value.WorkAreasInSync;
_tmpByte.4 := Value.SoftwareLimitsInSync;
_tmpByte.5 := Value.DefaultDynamicsInSync;
_tmpByte.6 := Value.ReferenceDynamicsInSync;
_tmpByte.7 := FALSE;

AddByte(_tmpByte);

AddDataInSync := PayloadLen;
END_METHOD

/// Adds a DWORD to the payload buffer , increase the payload pointer and returns the payload lenght
METHOD AddDword : UDINT
VAR_INPUT
  /// Value to add
  Value : DWORD;
END_VAR
// swap byte order
Value := SwapDword(Value);
// copy data 
SysDepMemCpy(pDest := ADR(Payload[PayloadPtr]), pSrc := ADR(Value), DataLen := SIZEOF(Value));
// inc data index 
PayloadPtr := PayloadPtr + SIZEOF(Value);
// return payload len
AddDword := PayloadLen := PayloadPtr;
END_METHOD

/// Adds two halfe BYTE to the payload buffer , increase the payload pointer and returns the payload lenght
METHOD AddHalfBytes : UDINT
VAR_INPUT
  /// Value to add
  HalfByteHi : BYTE;
  /// Value to add
  HalfByteLo : BYTE;
END_VAR

VAR
  /// internal value
 _value : BYTE;
END_VAR
_value := CombineHalfBytes( HalfByteHi := HalfByteHi, HalfByteLo := HalfByteLo);
// copy data 
SysDepMemCpy(pDest := ADR(Payload[PayloadPtr]), pSrc := ADR(_value), DataLen := SIZEOF(_value));
// inc payload pointer 
PayloadPtr := PayloadPtr + SIZEOF(_value);
// return payload len
AddHalfBytes := PayloadLen := PayloadPtr;
END_METHOD

/// Adds a IEC_DATE to the payload buffer, increase the payload pointer and returns the payload lenght
METHOD AddIecDate : UDINT
VAR_INPUT
  /// Value to add
  Value : IEC_DATE;
END_VAR
Value := SwapIecDate(Value);
// copy data 
SysDepMemCpy(pDest := ADR(Payload[PayloadPtr]), pSrc := ADR(Value), DataLen := SIZEOF(Value));
// inc payload pointer 
PayloadPtr := PayloadPtr + SIZEOF(Value);
// return payload len
AddIecDate := PayloadLen := PayloadPtr;
END_METHOD

/// Adds a IEC_TIME to the payload buffer, increase the payload pointer and returns the payload lenght
METHOD AddIecTime : UDINT
VAR_INPUT
  /// Value to add
  Value : IEC_TIME;
END_VAR
Value := SwapIecTime(Value);
// copy data 
SysDepMemCpy(pDest := ADR(Payload[PayloadPtr]), pSrc := ADR(Value), DataLen := SIZEOF(Value));
// inc payload pointer 
PayloadPtr := PayloadPtr + SIZEOF(Value);
// return payload len
AddIecTime := PayloadLen := PayloadPtr;
END_METHOD

/// Adds a INT to the payload buffer , increase the payload pointer and returns the payload lenght
METHOD AddInt : UDINT
VAR_INPUT
  /// Value to add
  Value : INT;
END_VAR
// swap byte order
Value := SwapInt(Value);
// copy data 
SysDepMemCpy(pDest := ADR(Payload[PayloadPtr]), pSrc := ADR(Value), DataLen := SIZEOF(Value));
// inc data index 
PayloadPtr := PayloadPtr + SIZEOF(Value);
// return payload len
AddInt := PayloadLen := PayloadPtr;
END_METHOD

/// Adds a REAL to the payload buffer , increase the payload pointer and returns the payload lenght
METHOD AddReal : UDINT
VAR_INPUT
  /// Value to add
  Value : REAL;
END_VAR
// swap byte order
Value := SwapReal(Value);
// copy data 
SysDepMemCpy(pDest := ADR(Payload[PayloadPtr]),pSrc := ADR(Value), DataLen := SIZEOF(Value));
// inc data index 
PayloadPtr := PayloadPtr + SIZEOF(Value);
// return payload len
AddReal := PayloadLen := PayloadPtr;
END_METHOD

/// Adds a SINT to the payload buffer, increase the payload pointer and returns the payload lenght
METHOD AddSint : UDINT
VAR_INPUT
  /// Value to add
  Value : SINT;
END_VAR
Value := Value;
// copy data 
SysDepMemCpy(pDest := ADR(Payload[PayloadPtr]), pSrc := ADR(Value), DataLen := SIZEOF(Value));
// inc payload pointer 
PayloadPtr := PayloadPtr + SIZEOF(Value);
// return payload len
AddSint := PayloadLen := PayloadPtr;
END_METHOD

/// Adds a String to the payload buffer, increase the payload pointer and returns the payload lenght
METHOD AddString : UDINT
VAR_INPUT
  /// Value to add
  Value : STRING(255);
END_VAR
IF ( LEN(Value) = 0 )
THEN
  RETURN;
END_IF

// copy data 
SysDepMemCpy(pDest := ADR(Payload[PayloadPtr]), pSrc := ADR(Value), DataLen := DINT_TO_UDINT(LEN(Value)));
// inc payload pointer 
PayloadPtr := PayloadPtr + DINT_TO_UDINT(LEN(Value));
// return payload len
AddString := PayloadLen := PayloadPtr;
END_METHOD

/// Adds a TIME to the payload buffer , increase the payload pointer and returns the payload lenght
METHOD AddTime : UDINT
VAR_INPUT
  /// Value to add
  Value : TOD;
END_VAR
// swap byte order
Value := SwapIecTime(Value);
// copy data 
SysDepMemCpy(pDest := ADR(Payload[PayloadPtr]), pSrc := ADR(Value), DataLen := SIZEOF(Value));
// inc data index 
PayloadPtr := PayloadPtr + SIZEOF(Value);
// return payload len
AddTime := PayloadLen := PayloadPtr;
END_METHOD

/// Adds a TurnNumber to the payload buffer, increase the payload pointer and returns the payload lenght
METHOD AddTurnNumber : UDINT
VAR_INPUT
  /// Value to add
  Value : TurnNumber;
END_VAR

VAR
  /// temporary Byte
 _tmpByte : BYTE;
END_VAR
Value := Value;

AddHalfBytes( HalfByteHi := SINT_TO_BYTE(Value.J2Turns) , HalfByteLo := SINT_TO_BYTE(Value.J1Turns));
AddHalfBytes( HalfByteHi := SINT_TO_BYTE(Value.J4Turns) , HalfByteLo := SINT_TO_BYTE(Value.J3Turns));
AddHalfBytes( HalfByteHi := SINT_TO_BYTE(Value.J6Turns) , HalfByteLo := SINT_TO_BYTE(Value.J5Turns));
AddByte(SINT_TO_BYTE(Value.E1Turns));

AddTurnNumber := PayloadLen;
END_METHOD

/// Adds a UDINT to the payload buffer , increase the payload pointer and returns the payload lenght
METHOD AddUdint : UDINT
VAR_INPUT
  /// Value to add
  Value : UDINT;
END_VAR
// swap byte order
Value := SwapUdint(Value);
// copy data 
SysDepMemCpy(pDest := ADR(Payload[PayloadPtr]), pSrc := ADR(Value), DataLen := SIZEOF(Value));
// inc data index 
PayloadPtr := PayloadPtr + SIZEOF(Value);
// return payload len
AddUdint := PayloadLen := PayloadPtr;
END_METHOD

/// Adds a UINT to the payload buffer , increase the payload pointer and returns the payload lenght
METHOD AddUint : UDINT
VAR_INPUT
  /// Value to add
  Value : UINT;
END_VAR
// swap byte order
Value := SwapUint(Value);
// copy data 
SysDepMemCpy(pDest := ADR(Payload[PayloadPtr]), pSrc := ADR(Value), DataLen := SIZEOF(Value));
// inc data index 
PayloadPtr := PayloadPtr + SIZEOF(Value);
// return payload len
AddUint := PayloadLen := PayloadPtr;
END_METHOD

/// Adds a USINT to the payload buffer, increase the payload pointer and returns the payload lenght
METHOD AddUsint : UDINT
VAR_INPUT
  /// Value to add
  Value : USINT;
END_VAR
Value := Value;
// copy data 
SysDepMemCpy(pDest := ADR(Payload[PayloadPtr]), pSrc := ADR(Value), DataLen := SIZEOF(Value));
// inc payload pointer 
PayloadPtr := PayloadPtr + SIZEOF(Value);
// return payload len
AddUsint := PayloadLen := PayloadPtr;
END_METHOD

/// Resets the payload buffer, the payload pointer and the payload length
METHOD Reset
VAR_INPUT
END_VAR
SysDepMemSet(pDest := ADR(Payload), Value := 0 , DataLen := SIZEOF(Payload));
PayloadLen := 0;
PayloadPtr := 0;
END_METHOD

END_FUNCTION_BLOCK

// Library/POUs/_internal/ActiveCommandRegisterFB
FUNCTION_BLOCK ActiveCommandRegisterFB EXTENDS RobotLibraryLogFB
// ------------------------------------------------------------------------- 
//  SRCI Robot Library                                                
// ------------------------------------------------------------------------- 
//                                                                           
//  Object:      ActiveCommandRegisterFB                                       
//  Author:      Thorsten Brach                                                
//  Date:        2024-06-01
//
//  Description:                                              
//   
//                                                                           
//  Copyright: 
//    (C) 2024 Thorsten Brach. All rights reserved                                                                                                                                            
//             Licensed under the LGPL-3.0 license.
//                                                                           
//  Disclaimer:                                                                           
//    This project is provided without any guarantee and can be used for   
//    private and commercial purposes. Any use is at the user’s 
//    own risk and responsibility.
//
// -------------------------------------------------------------------------
VAR_INPUT
  /// Active Command Register
  Register            : ARRAY [1..RobotLibraryParameter.ACTIVE_CMD_REGISTER_ENTRIES_MAX] OF AxesGroupAcyclicAcrEntry;
  /// System Time
  SystemTime          : SystemTime;
  /// usable size of the arc register
  RegisterSize        : DINT := RobotLibraryParameter.ACTIVE_CMD_REGISTER_ENTRIES_MAX;
END_VAR

VAR_OUTPUT
  /// Execution Order List 
  ExecutionOrderList  : ARRAY [1..RobotLibraryParameter.ACTIVE_CMD_REGISTER_ENTRIES_MAX] OF DINT;
END_VAR


VAR
  /// temporarty Active Command Register
  TmpRegister        : ARRAY [1..RobotLibraryParameter.ACTIVE_CMD_REGISTER_ENTRIES_MAX] OF AxesGroupAcyclicAcrEntry;
  /// last used unique ID 
  LastUniqueID       : UINT;
  ///
  
END_VAR

VAR CONSTANT
  /// Active command
  ACTIVE_CMD           : UDINT := 1;
  /// Buffered command
  BUFFER_CMD           : UDINT := 2;
  /// Empty ARC entry
  EMPTY_ARC_ENTRY      : AxesGroupAcyclicAcrEntry := (State := ActiveCommandRegisterState.IS_FREE);
  /// Empty command entry
  EMPTY_CMD_ENTRY      : AxesGroupAcyclicAcrEntryCmdBuffer := (State := BufferStateCmd.EMPTY);
  
  /// constant for byte index of priority in payload 
  PRIORITY_IDX         : BYTE := 3;  /// bitmask to mask the priority out of the halfbyte
  PRIORITY_BIT_MASK    : BYTE := 2#000_1111;   
END_VAR

ManageRegister();

UpdateExecutionOrderList();

METHOD PUBLIC AddCmd : UDINT
VAR_INPUT
  /// Pointer to the corresponding command-FB to enable a callback mechanism
  pCommandFB   : POINTER TO RobotLibraryBaseFB;
END_VAR

VAR
  /// internal index for loops
 _regIdx     : DINT;
  /// internal command type 
 _cmdType    : CmdType;
  /// log message
 _messageLog : AlarmMessage;  
END_VAR
// calculate the used length of the ARC 
FOR _regIdx := 1 TO RegisterSize
DO
  IF ( Register[_regIdx].State = ActiveCommandRegisterState.IS_FREE )
  THEN
    Register[_regIdx].State                        := ActiveCommandRegisterState.IS_PROCESSING;
    //Register[_regIdx].UniqueID                     := CreateUniqueID();
    Register[_regIdx].UniqueID                     := DINT_TO_UINT(_regIdx);
    Register[_regIdx].pCommandFB                   := pCommandFB;

    // check pointer to command FB
    IF ( Register[_regIdx].pCommandFB <> RobotLibraryConstants.NULL_POINTER )
    THEN
      Register[_regIdx].Command[RobotLibraryConstants.ACTIVE_CMD].Timestamp  := SystemTime;
      Register[_regIdx].Command[RobotLibraryConstants.ACTIVE_CMD].Payload    := pCommandFB^.CommandData.Payload;
      Register[_regIdx].Command[RobotLibraryConstants.ACTIVE_CMD].PayloadLen := pCommandFB^.CommandData.PayloadLen;
      Register[_regIdx].Command[RobotLibraryConstants.ACTIVE_CMD].PayLoadPtr := 0;
      Register[_regIdx].Command[RobotLibraryConstants.ACTIVE_CMD].State      := BufferStateCmd.CREATED;
    END_IF
  
    // return Unique ID
    AddCmd := Register[_regIdx].UniqueID;

    // Get CmdType from payload
    SysDepMemCpy( pDest := ADR(_cmdType), pSrc := ADR(pCommandFB^.CommandData.Payload), DataLen := SIZEOF(_cmdType));
    
    // Create log entry
    CreateLogMessagePara1 ( Timestamp   := SystemTime,
                            MessageType := MessageType.CMD,
                            Severity    := Severity.DEBUG,
                            MessageCode := 0,
                            MessageText := 'Added Cmd <{1}> to active command register',
                            Para1       :=  CMD_TYPE_TO_STRING(SwapUint(_cmdType)));
    EXIT;
  END_IF
END_FOR
END_METHOD

METHOD AddRsp : UDINT
VAR_INPUT
  /// Response
  Rsp : TelegramRobToPlcFragment;
END_VAR
VAR
  /// internal index for loops
 _Idx             : DINT;
  /// internal registen index
 _regIdx          : DINT;
  /// internal command type
 _cmdType         : CmdType;
  /// internal FragmentAction
 _fragmentAction  :  FragmentAction;
  /// internal command message state
 _cmdMessageState : CmdMessageState;
  /// internal flag for CmdID found
 _found           : BOOL;
END_VAR
FOR _regIdx := 1 TO RegisterSize
DO
  IF ( Register[_regIdx].UniqueID = Rsp.Header.CmdID )
  THEN
    // CmdID was found in the ARC
   _found := TRUE;
    // convert to fragment action 
   _fragmentAction := ByteToFragmentAction(Rsp.Header.FragmentAction);

    // delete response 
    IF ( _fragmentAction.Clear )
    THEN
      SysDepMemSet( pDest := ADR(Register[_regIdx].Response[1]), Value := 0, DataLen := SIZEOF(Register[_regIdx].Response[1]));
    END_IF
                       
    // add payload to response
    FOR _idx := Rsp.Header.PayloadPointer TO  Rsp.Header.PayloadLength -1
    DO
      Register[_regIdx].Response[1].Timestamp     := SystemTime;
      Register[_regIdx].Response[1].State         := BufferStateRsp.RECEIVING;
      Register[_regIdx].Response[1].PayloadLen    := Register[_regIdx].Response[1].PayloadLen + 1;
      Register[_regIdx].Response[1].Payload[_idx] := Rsp.Command.Payload[_idx];
    END_FOR

    // Get current message state 
   _cmdMessageState := GetHalfeByteLo    (Value  := Register[_regIdx].Response[ACTIVE_CMD].Payload[0]);
    // Get command type from payload
   _cmdType         := CombineBytesToUint(HiByte := Register[_regIdx].Command [ACTIVE_CMD].Payload[0],
                                          LoByte := Register[_regIdx].Command [ACTIVE_CMD].Payload[1]);

    // Create log entry
    CreateLogMessagePara3 ( Timestamp   := SystemTime,
                            MessageType := MessageType.CMD,
                            Severity    := Severity.DEBUG,
                            MessageCode := 0,
                            MessageText := 'Added Response of CmdID <{1}>, CmdType <{2}> with State = {3} to ACR',
                            Para1       :=  UINT_TO_STRING(Rsp.Header.CmdID),
                            Para2       :=  CMD_TYPE_TO_STRING(_cmdType),
                            Para3       :=  CMD_MESSAGE_STATE_TO_STRING(_cmdMessageState));

    IF ( _fragmentAction.Complete )
    THEN
      // set response state
      Register[_regIdx].Response[1].State := BufferStateRsp.RECEIVED;      
     
      // Check current message state and tag the register state as IS_FINAL, if needed 
      IF ( _cmdMessageState >= CmdMessageState.DONE) 
      THEN
        Register[_regIdx].State := ActiveCommandRegisterState.IS_FINAL;
        
        // get command type from payload
       _cmdType := CombineBytesToUint(HiByte := Register[_regIdx].Command[ACTIVE_CMD].Payload[0],
                                      LoByte := Register[_regIdx].Command[ACTIVE_CMD].Payload[1]);

        // Create log entry
        CreateLogMessagePara3( Timestamp   := SystemTime,
                               MessageType := MessageType.CMD,
                               Severity    := Severity.DEBUG,
                               MessageCode := 0,
                               MessageText := 'ARC Register [{1}] : Response of CmdID <{2}>, CmdType <{3}> has reached Final State',
                               Para1       :=  DINT_TO_STRING(_regIdx),
                               Para2       :=  UINT_TO_STRING(Rsp.Header.CmdID),
                               Para3       :=  CMD_TYPE_TO_STRING(_cmdType));
                               
        // Exit the loop
      END_IF      
    END_IF
    
    EXIT;
  END_IF
END_FOR


// Check CmdID was found in the ARC ? 
IF ( NOT _found )
THEN
  // Create log entry
  CreateLogMessagePara2 ( Timestamp   := SystemTime,
                          MessageType := MessageType.CMD,
                          Severity    := Severity.WARNING,
                          MessageCode := 0,
                          MessageText := 'Rsp <{1}> with State = {2} received, but no matching ARC entry found',
                          Para1       :=  UINT_TO_STRING(Rsp.Header.CmdID),
                          Para2       :=  CMD_MESSAGE_STATE_TO_STRING(_cmdMessageState));
END_IF
END_METHOD

METHOD PRIVATE CreateUniqueID : UINT
VAR
  /// internal index for loops
 _idx : DINT;
  /// length of the ARC
 _arcLenght : DINT;
END_VAR
// inc last unique ID 
LastUniqueID := LastUniqueID + 1;
// return unique ID
CreateUniqueID := LastUniqueID;
END_METHOD

METHOD FB_init : BOOL
VAR_INPUT
  bInitRetains : BOOL; // if TRUE, the retain variables are initialized (warm start / cold start)
  bInCopyCode : BOOL;  // if TRUE, the instance afterwards gets moved into the copy code (online change)
END_VAR
MyType := 'ActiveCommandRegisterFB';
END_METHOD

METHOD PRIVATE ManageRegister
VAR
  /// internal index
 _regIdx     : DINT;
  /// internal command type
 _cmdType    : CmdType;
END_VAR
FOR _regIdx := 1 TO RegisterSize
DO
  // Check pointer to command FB is valid ? 
  IF ( Register[_regIdx].pCommandFB = RobotLibraryConstants.NULL_POINTER)
  THEN
    RETURN;
  END_IF

  // Check apply Cmd parameter update ?  
  IF (( Register[_regIdx].Command[ACTIVE_CMD].State = BufferStateCmd.PROCESSED        ) AND
      ( Register[_regIdx].Command[BUFFER_CMD].State = BufferStateCmd.UPDATE_AVAILABLE ))
  THEN
    Register[_regIdx].Command[ACTIVE_CMD] := Register[_regIdx].Command[BUFFER_CMD];
    Register[_regIdx].Command[BUFFER_CMD] := EMPTY_CMD_ENTRY;

    // get command type from payload
   _cmdType := CombineBytesToUint(HiByte := Register[_regIdx].Command[ACTIVE_CMD].Payload[0],
                                  LoByte := Register[_regIdx].Command[ACTIVE_CMD].Payload[1]);

    // Create log entry
    CreateLogMessagePara3 ( Timestamp   := SystemTime,
                            MessageType := MessageType.CMD,
                            Severity    := Severity.DEBUG,
                            MessageCode := 0,
                            MessageText := 'ARC Register [{1}] : Moved BUFFER_CMD to ACTIVE_CMD, CmdID <{2}> , CmdType <{3}>',
                            Para1       :=  DINT_TO_STRING(_regIdx),
                            Para2       :=  UINT_TO_STRING(Register[_regIdx].UniqueID),
                            Para3       :=  CMD_TYPE_TO_STRING(_cmdType));

  END_IF
  
  // Check Response received ? 
  IF ( Register[_regIdx].Response[ACTIVE_CMD].State = BufferStateRsp.RECEIVED)
  THEN
    // update state
    Register[_regIdx].Response[ACTIVE_CMD].State := BufferStateRsp.PROCESSED;
    // callback CommandFB    
    Register[_regIdx].pCommandFB^.CallBack(RspData := Register[_regIdx].Response[ACTIVE_CMD],TimeStamp := SystemTime);    
  END_IF

  // delete entries with State.IS_Final 
  IF ( Register[_regIdx].State = ActiveCommandRegisterState.IS_FINAL )
  THEN
  
    // get command type from payload
   _cmdType := CombineBytesToUint(HiByte := Register[_regIdx].Command[ACTIVE_CMD].Payload[0],
                                  LoByte := Register[_regIdx].Command[ACTIVE_CMD].Payload[1]);

    // Create log entry
    CreateLogMessagePara3( Timestamp   := SystemTime,
                           MessageType := MessageType.CMD,
                           Severity    := Severity.DEBUG,
                           MessageCode := 0,
                           MessageText := 'ARC Register [{1}} : Deleted CmdID <{2}> , CmdType <{3}> from ARC, because of Final-State was reached',
                           Para1       :=  DINT_TO_STRING(_regIdx),
                           Para2       :=  UINT_TO_STRING(Register[_regIdx].UniqueID),  
                           Para3       :=  CMD_TYPE_TO_STRING(_cmdType));

                           
    Register[_regIdx] := EMPTY_ARC_ENTRY;                           
  END_IF
 
END_FOR
END_METHOD

PROPERTY PUBLIC NotifyParameterChanged : UDINT
SET
VAR
  /// internal register index
 _regIdx : DINT;
END_VAR
FOR _regIdx := 1 TO RobotLibraryParameter.ACTIVE_CMD_REGISTER_ENTRIES_MAX
DO
  // check unique ID found ?
  IF ( Register[_regIdx].UniqueID = NotifyParameterChanged )
  THEN  
    IF (( Register[_regIdx].Command[ACTIVE_CMD].State <> BufferStateCmd.SENDING   ) AND
        ( Register[_regIdx].Command[ACTIVE_CMD].State <> BufferStateCmd.PROCESSED ))
    THEN
      // Check pointer is valid ? 
      IF ( Register[_regIdx].pCommandFB <> RobotLibraryConstants.NULL_POINTER )
      THEN
        // add to send register
        Register[_regIdx].Command[ACTIVE_CMD].Timestamp  := SystemTime;
        Register[_regIdx].Command[ACTIVE_CMD].State      := BufferStateCmd.UPDATE_AVAILABLE;
        Register[_regIdx].Command[ACTIVE_CMD].Payload    := Register[_regIdx].pCommandFB^.CommandData.Payload;
        Register[_regIdx].Command[ACTIVE_CMD].PayloadLen := Register[_regIdx].pCommandFB^.CommandData.PayloadLen;

        // Create log entry
        CreateLogMessagePara2 ( Timestamp   := SystemTime,
                                MessageType := MessageType.CMD,
                                Severity    := Severity.DEBUG,
                                MessageCode := 0,
                                MessageText := 'Parameter update from {1} with CmdID <{2}> received -> written to ACTIVE_CMD Index',
                                Para1       :=  Register[_regIdx].pCommandFB^.MyType,
                                Para2       :=  UDINT_TO_STRING(NotifyParameterChanged));
      END_IF
    ELSE
      // Check pointer is valid ? 
      IF ( Register[_regIdx].pCommandFB <> RobotLibraryConstants.NULL_POINTER )
      THEN
        // add to buffer register
        Register[_regIdx].Command[BUFFER_CMD].Timestamp  := SystemTime;
        Register[_regIdx].Command[BUFFER_CMD].State      := BufferStateCmd.UPDATE_AVAILABLE;
        Register[_regIdx].Command[BUFFER_CMD].Payload    := Register[_regIdx].pCommandFB^.CommandData.Payload;
        Register[_regIdx].Command[BUFFER_CMD].PayloadLen := Register[_regIdx].pCommandFB^.CommandData.PayloadLen;

        // Create log entry
        CreateLogMessagePara2 ( Timestamp   := SystemTime,
                                MessageType := MessageType.CMD,
                                Severity    := Severity.DEBUG,
                                MessageCode := 0,
                                MessageText := 'Parameter update from {1} with CmdID <{2}> received -> written to BUFFER_CMD Index',
                                Para1       :=  Register[_regIdx].pCommandFB^.MyType,
                                Para2       :=  UDINT_TO_STRING(NotifyParameterChanged));
      END_IF
    END_IF
    
    
  END_IF
END_FOR
END_SET
END_PROPERTY

METHOD PUBLIC OnOnlineChange : DINT
VAR_INPUT
  /// unique ID 
  UniqueID     : UDINT;
  /// Pointer to the corresponding command-FB to enable a callback mechanism
  pCommandFB   : POINTER TO RobotLibraryBaseFB;
END_VAR

VAR
  /// internal index for loops
 _regIdx : DINT;
END_VAR
OnOnlineChange := -1;

// Check command FB pointer is valid ?
IF ( pCommandFB <> RobotLibraryConstants.NULL_POINTER)
THEN
  FOR _regIdx := 1 TO RegisterSize
  DO
    // check unique ID found ?
    IF ( Register[_regIdx].UniqueID = UniqueID ) 
    THEN  
      // update pointer to command FB
      Register[_regIdx].pCommandFB := pCommandFB;
      // Return result OK
      OnOnlineChange := RobotLibraryConstants.OK;
      EXIT;
    END_IF
  END_FOR
END_IF
END_METHOD

METHOD PUBLIC RemoveCmd
VAR_INPUT
 /// unique ID
 UniqueID : UDINT;  
END_VAR

VAR
  /// internal index
 _regIdx : DINT;
END_VAR
FOR _regIdx := 1 TO RegisterSize
DO
  // check unique ID found and not yet sended ?
  IF (( Register[_regIdx].UniqueID         = UniqueID               ) AND
      ( Register[_regIdx].Command[1].State < BufferStateCmd.SENDING ))       
  THEN  
    // delete register entry
    SysDepMemSet(pDest := ADR(Register[_regIdx]), Value := 0 , DataLen := SIZEOF(Register[_regIdx]));
    EXIT;
  END_IF
END_FOR
END_METHOD

METHOD PRIVATE UpdateExecutionOrderList
VAR
  /// temporary Active Command Register entry
  TmpRegisterEntry : AxesGroupAcyclicAcrEntry;
  /// temporary index
  TmpIndex         : DINT;
  /// internal index
  i                : DINT;  
  /// internal index
  j                : DINT;  
END_VAR
// Reset temporary register
SysDepMemSet(pDest := ADR(TmpRegister)       , Value := 0, DataLen := SIZEOF(TmpRegister));
// Reset Execution Order List
SysDepMemSet(pDest := ADR(ExecutionOrderList), Value := 0, DataLen := SIZEOF(ExecutionOrderList));
// pre-set temporary register index 
j := 1;

FOR i := 1 TO RegisterSize
DO
  // add only entries which are not in status free and where datas must be processed
  IF (( Register[i].State                      > ActiveCommandRegisterState.IS_FREE ) AND
      ( Register[i].Command[ACTIVE_CMD].State <> BufferStateCmd.EMPTY               ) AND
      ( Register[i].Command[ACTIVE_CMD].State <> BufferStateCmd.PROCESSED           ))
  THEN
    // copy register entry 
    TmpRegister[j] := Register[i];
    // store index of the entry from the ARC
    ExecutionOrderList[j] := i;
    // inc temporar register index
    j := j + 1; 
  END_IF
END_FOR  

// Bubble Sort to sort the priorities from the active command register
FOR i := 1 TO RegisterSize
DO
  FOR j := 1 TO RegisterSize - 1
  DO 
    // check list entry is not empty ? 
    IF (( TmpRegister[i  ].State = ActiveCommandRegisterState.IS_FREE ) OR
        ( TmpRegister[j+1].State = ActiveCommandRegisterState.IS_FREE ))
    THEN
      EXIT; 
    END_IF  

    IF (( TmpRegister[j].Command[ACTIVE_CMD].Payload[PRIORITY_IDX] AND PRIORITY_BIT_MASK ) > ( TmpRegister[j+1].Command[ACTIVE_CMD].Payload[PRIORITY_IDX] AND PRIORITY_BIT_MASK ))
    THEN    
      // swap position of register entry  
      TmpRegisterEntry := TmpRegister[j];         
      TmpRegister[j]   := TmpRegister[j+1];
      TmpRegister[j+1] := TmpRegisterEntry;
      
      // swap position of index in the Execution Order List  
      TmpIndex                := ExecutionOrderList[j];
      ExecutionOrderList[j]   := ExecutionOrderList[j+1];
      ExecutionOrderList[j+1] := TmpIndex;
    END_IF
  END_FOR 
END_FOR

// Bubble Sort to sort the Timestamp from the pre-sorted active command register
FOR i := 1 TO RegisterSize
DO
  FOR j := 1 TO RegisterSize - 1
  DO    
    // check list entry is not empty ? 
    IF (( TmpRegister[i  ].State = ActiveCommandRegisterState.IS_FREE ) OR
        ( TmpRegister[j+1].State = ActiveCommandRegisterState.IS_FREE ))
    THEN
      EXIT; 
    END_IF  

       // Priority is higher
    IF (( TmpRegister[j].Command[ACTIVE_CMD].Payload[PRIORITY_IDX] AND PRIORITY_BIT_MASK ) >= ( TmpRegister[j+1].Command[ACTIVE_CMD].Payload[PRIORITY_IDX] AND PRIORITY_BIT_MASK )) AND
       // Date is greater 
       (( TmpRegister[j].Command[ACTIVE_CMD].Timestamp.SystemDate                          >    TmpRegister[j+1].Command[ACTIVE_CMD].Timestamp.SystemDate                         ) OR 
       // Date is the same, but Time is greater
       (( TmpRegister[j].Command[ACTIVE_CMD].Timestamp.SystemDate                          =    TmpRegister[j+1].Command[ACTIVE_CMD].Timestamp.SystemDate                         ) AND 
        ( TmpRegister[j].Command[ACTIVE_CMD].Timestamp.SystemTime                          >    TmpRegister[j+1].Command[ACTIVE_CMD].Timestamp.SystemTime                         )))
    THEN    
      // swap position of register entry  
      TmpRegisterEntry := TmpRegister[j];         
      TmpRegister[j]   := TmpRegister[j+1];
      TmpRegister[j+1] := TmpRegisterEntry;
      
      // swap position of index in the Execution Order List  
      TmpIndex                := ExecutionOrderList[j];
      ExecutionOrderList[j]   := ExecutionOrderList[j+1];
      ExecutionOrderList[j+1] := TmpIndex;
    END_IF
  END_FOR 
END_FOR
END_METHOD

END_FUNCTION_BLOCK

// Library/POUs/_internal/RobotLibraryLogFB
FUNCTION_BLOCK RobotLibraryLogFB
// ------------------------------------------------------------------------- 
//  SRCI Robot Library                                                
// ------------------------------------------------------------------------- 
//                                                                           
//  Object:      RobotLibraryLogFB                                       
//  Author:      Thorsten Brach                                                
//  Date:        2024-11-10
//
//  Description:                                              
//   
//                                                                           
//  Copyright: 
//    (C) 2024 Thorsten Brach. All rights reserved                                                                                                                                            
//             Licensed under the LGPL-3.0 license.
//                                                                           
//  Disclaimer:                                                                           
//    This project is provided without any guarantee and can be used for   
//    private and commercial purposes. Any use is at the user’s 
//    own risk and responsibility.
//
// -------------------------------------------------------------------------
VAR_INPUT
  /// Interface to an external logger
  ExternalLogger : IMessageLogger;  
  /// Logging level
  LogLevel       : LogLevelEnum := LogLevelEnum.INFO; 
END_VAR

VAR
  /// Type of the function block
 _myType         : STRING;
END_VAR

METHOD CreateLogMessage
VAR_INPUT
  /// Timestamp
  Timestamp   : SystemTime;
  /// Type of message according to Table 5-46:
  MessageType : MessageType;
  /// Severity of message according to Table 5-47: Debug, Info, Warning, Error, Fatal error
  Severity    : Severity;
  /// Code of messages
  MessageCode : DWORD;
  /// Static text of message
  MessageText : STRING(255);  
END_VAR

VAR
  /// internal log message 
 _logMessage : AlarmMessage;
END_VAR
IF (( ExternalLogger <> 0        ) AND 
    ( LogLevel       <= Severity )) {warning 'ToDo: LogLevel and Severity are the same -> use an alias for it'}
THEN
 _logMessage.Timestamp   := Timestamp;
 _logMessage.MessageType := MessageType;
 _logMessage.Severity    := Severity;
 _logMessage.MessageCode := MessageCode;
 _logMessage.MessageText := StrPadRight(MyType,' ', RobotLibraryDefines.MaxTypeNameLength);
 _logMessage.MessageText := CONCAT(_logMessage.MessageText, ': ');
 _logMessage.MessageText := CONCAT(_logMessage.MessageText,MessageText);
  
  ExternalLogger.AddMessageLog( _logMessage);
END_IF
END_METHOD

METHOD CreateLogMessagePara1
VAR_INPUT
  /// Timestamp
  Timestamp   : SystemTime;
  /// Type of message according to Table 5-46:
  MessageType : MessageType;
  /// Severity of message according to Table 5-47: Debug, Info, Warning, Error, Fatal error
  Severity    : Severity;
  /// Code of messages
  MessageCode : DWORD;
  /// Static text of message
  MessageText : STRING(255);  
  /// sub string which will replace the placeholder {1}
  Para1       : STRING(255);
END_VAR
VAR
  /// internal log message 
 _logMessage : AlarmMessage;
END_VAR
MessageText := StrReplace(MessageText,'{1}', Para1);

CreateLogMessage( Timestamp   := Timestamp,
                  MessageType := MessageType,
                  Severity    := Severity,
                  MessageCode := MessageCode,
                  MessageText := MessageText);
END_METHOD

METHOD CreateLogMessagePara2 : BOOL
VAR_INPUT
  /// Timestamp
  Timestamp   : SystemTime;
  /// Type of message according to Table 5-46:
  MessageType : MessageType;
  /// Severity of message according to Table 5-47: Debug, Info, Warning, Error, Fatal error
  Severity    : Severity;
  /// Code of messages
  MessageCode : DWORD;
  /// Static text of message
  MessageText : STRING(255);  
  /// sub string which will replace the placeholder {1}
  Para1       : STRING(255);
  /// sub string which will replace the placeholder {2}
  Para2       : STRING(255);
END_VAR
VAR
  /// internal log message 
 _logMessage : AlarmMessage;
END_VAR
MessageText := StrReplace(MessageText,'{2}', Para2);

CreateLogMessagePara1( Timestamp   := Timestamp,
                       MessageType := MessageType,
                       Severity    := Severity,
                       MessageCode := MessageCode,
                       MessageText := MessageText,
                       Para1       := Para1);
END_METHOD

METHOD CreateLogMessagePara3
VAR_INPUT
  /// Timestamp
  Timestamp   : SystemTime;
  /// Type of message according to Table 5-46:
  MessageType : MessageType;
  /// Severity of message according to Table 5-47: Debug, Info, Warning, Error, Fatal error
  Severity    : Severity;
  /// Code of messages
  MessageCode : DWORD;
  /// Static text of message
  MessageText : STRING(255);  
  /// sub string which will replace the placeholder {1}
  Para1       : STRING(255);
  /// sub string which will replace the placeholder {2}
  Para2       : STRING(255);
  /// sub string which will replace the placeholder {3}
  Para3       : STRING(255);
END_VAR
VAR
  /// internal log message 
 _logMessage : AlarmMessage;
END_VAR
MessageText := StrReplace(MessageText,'{3}', Para3);

CreateLogMessagePara2( Timestamp   := Timestamp,
                       MessageType := MessageType,
                       Severity    := Severity,
                       MessageCode := MessageCode,
                       MessageText := MessageText,
                       Para1       := Para1,
                       Para2       := Para2);
END_METHOD

METHOD CreateLogMessagePara4 : BOOL
VAR_INPUT
  /// Timestamp
  Timestamp   : SystemTime;
  /// Type of message according to Table 5-46:
  MessageType : MessageType;
  /// Severity of message according to Table 5-47: Debug, Info, Warning, Error, Fatal error
  Severity    : Severity;
  /// Code of messages
  MessageCode : DWORD;
  /// Static text of message
  MessageText : STRING(255);  
  /// sub string which will replace the placeholder {1}
  Para1       : STRING(255);
  /// sub string which will replace the placeholder {2}
  Para2       : STRING(255);
  /// sub string which will replace the placeholder {3}
  Para3       : STRING(255);
  /// sub string which will replace the placeholder {4}
  Para4       : STRING(255);
END_VAR
VAR
  /// internal log message 
 _logMessage : AlarmMessage;
END_VAR
MessageText := StrReplace(MessageText,'{4}', Para4);

CreateLogMessagePara3( Timestamp   := Timestamp,
                       MessageType := MessageType,
                       Severity    := Severity,
                       MessageCode := MessageCode,
                       MessageText := MessageText,
                       Para1       := Para1,
                       Para2       := Para2,
                       Para3       := Para3);
END_METHOD

METHOD CreateLogMessagePara5 
VAR_INPUT
  /// Timestamp
  Timestamp   : SystemTime;
  /// Type of message according to Table 5-46:
  MessageType : MessageType;
  /// Severity of message according to Table 5-47: Debug, Info, Warning, Error, Fatal error
  Severity    : Severity;
  /// Code of messages
  MessageCode : DWORD;
  /// Static text of message
  MessageText : STRING(255);  
  /// sub string which will replace the placeholder {1}
  Para1       : STRING(255);
  /// sub string which will replace the placeholder {2}
  Para2       : STRING(255);
  /// sub string which will replace the placeholder {3}
  Para3       : STRING(255);
  /// sub string which will replace the placeholder {4}
  Para4       : STRING(255);
  /// sub string which will replace the placeholder {5}
  Para5       : STRING(255);
END_VAR
VAR
  /// internal log message 
 _logMessage : AlarmMessage;
END_VAR
MessageText := StrReplace(MessageText,'{5}', Para5);

CreateLogMessagePara4( Timestamp   := Timestamp,
                       MessageType := MessageType,
                       Severity    := Severity,
                       MessageCode := MessageCode,
                       MessageText := MessageText,
                       Para1       := Para1,
                       Para2       := Para2,
                       Para3       := Para3,
                       Para4       := Para4);
END_METHOD

METHOD CreateLogMessagePara6 
VAR_INPUT
  /// Timestamp
  Timestamp   : SystemTime;
  /// Type of message according to Table 5-46:
  MessageType : MessageType;
  /// Severity of message according to Table 5-47: Debug, Info, Warning, Error, Fatal error
  Severity    : Severity;
  /// Code of messages
  MessageCode : DWORD;
  /// Static text of message
  MessageText : STRING(255);  
  /// sub string which will replace the placeholder {1}
  Para1       : STRING(255);
  /// sub string which will replace the placeholder {2}
  Para2       : STRING(255);
  /// sub string which will replace the placeholder {3}
  Para3       : STRING(255);
  /// sub string which will replace the placeholder {4}
  Para4       : STRING(255);
  /// sub string which will replace the placeholder {5}
  Para5       : STRING(255);
  /// sub string which will replace the placeholder {6}
  Para6       : STRING(255);
END_VAR
VAR
  /// internal log message 
 _logMessage : AlarmMessage;
END_VAR
MessageText := StrReplace(MessageText,'{6}', Para6);

CreateLogMessagePara5( Timestamp   := Timestamp,
                       MessageType := MessageType,
                       Severity    := Severity,
                       MessageCode := MessageCode,
                       MessageText := MessageText,
                       Para1       := Para1,
                       Para2       := Para2,
                       Para3       := Para3,
                       Para4       := Para4,
                       Para5       := Para5);
END_METHOD

PROPERTY PROTECTED MyType : STRING
GET
MyType := _myType;
END_GET
SET
_myType := MyType;

// set the max type name length 
RobotLibraryDefines.MaxTypeNameLength := MAX(LEN(_myType), RobotLibraryDefines.MaxTypeNameLength);
END_SET
END_PROPERTY

END_FUNCTION_BLOCK

// Library/POUs/_internal/RobotLibraryBaseFB
FUNCTION_BLOCK RobotLibraryBaseFB EXTENDS RobotLibraryLogFB
// ------------------------------------------------------------------------- 
//  SRCI Robot Library                                                
// ------------------------------------------------------------------------- 
//                                                                           
//  Object:      RobotLibraryBaseFB                                       
//  Author:      Thorsten Brach                                                
//  Date:        2024-06-01
//
//  Description:                                              
//   
//                                                                           
//  Copyright: 
//    (C) 2024 Thorsten Brach. All rights reserved                                                                                                                                            
//             Licensed under the LGPL-3.0 license.
//                                                                           
//  Disclaimer:                                                                           
//    This project is provided without any guarantee and can be used for   
//    private and commercial purposes. Any use is at the user’s 
//    own risk and responsibility.
//
// -------------------------------------------------------------------------
VAR_INPUT
  /// User defined command name
  Name         : STRING(20);
  /// Execution Mode
  ExecMode     : ExecutionMode;
  /// Priority
  Priority     : PriorityLevel;
END_VAR
VAR_OUTPUT
  /// Command data
  CommandData  : RobotLibrarySendDataFB;
  /// response data
  ResponseData : RobotLibraryRecvDataFB;
  /// An error occurred during the execution of the command
  Error        : BOOL;
  /// ErrorID reported by RC for error identification according to Table 7-1
  ErrorID      : WORD;
  ErrorIdEnum  : RobotLibraryErrorIdEnum;  
  ErrorAddTxt  : STRING(RobotLibraryConstants.MAX_ADD_TEXT_LENGTH);
  
  /// WarningID for warning identification reported during execution of command according to Table 7-3
  WarningID    : WORD;
  WarningIdEnum: RobotLibraryWarningIdEnum;  
  /// InfoID for info identification reported during execution of command according to Table 7-5
  InfoID       : WORD;    
  InfoIdEnum   : RobotLibraryInfoIdEnum;  
END_VAR
VAR_IN_OUT
  /// Robot assignment of function
  AxesGroup    : AxesGroup; 
END_VAR

VAR
  /// Rising edge for error
 _error_R                  : R_TRIG;
  /// Rising edge for warning
 _warning_R                : R_TRIG;
  /// Rising edge for information
 _info_R                   : R_TRIG;
  /// unique ID
 _uniqueID                 : UDINT;  
  /// flag for response received
 _responseReceived         : BOOL;
  /// internal step counter
 _stepCmd                  : DINT;
  /// internal timer  
 _timerCmd                 : TON;
  /// internal timeout 
 _timeoutCmd               : TIME := T#5S;
  /// internal command header
 _cmdHeader                : CmdHeader;  
  /// internal response header
 _rspHeader                : RspHeader;
  /// internal flag for send a parameter update
 _parameterUpdateInternal  : BOOL; 
  /// internal flag for parameter has changed
 _parameterChanged         : BOOL;
  /// internal flag for parameter are valid
 _parameterValid           : BOOL;
END_VAR

OnCall               (AxesGroup := AxesGroup);
CheckParameterChanged(AxesGroup := AxesGroup);


IF ( AxesGroup.InternalData.OnlineChange_R.Q )
THEN
  OnOnlineChange(AxesGroup := AxesGroup);
END_IF

